// TwinCAT 3 PLC project Sample02
// ProgramVersion: 3.1.0.8
// libraries:
//   Tc2_Standard, * (Beckhoff Automation GmbH)
//   Tc2_System, * (Beckhoff Automation GmbH)
//   Tc2_Utilities, * (Beckhoff Automation GmbH)
//   Tc3_Interfaces, * (Beckhoff Automation GmbH)
//   Tc3_MemMan, * (Beckhoff Automation GmbH)
//   Tc3_Module, * (Beckhoff Automation GmbH)
// project tree:
//   / PlcTask.TcTTO (not stored)
//   POUs/ FB_AbstractLoggerFactory.TcPOU (not stored), FB_CsvLogger.TcPOU (not stored), FB_FileLoggerFactory.TcPOU, FB_Logger.TcPOU, FB_TxtLogger.TcPOU (not stored), FB_XmlLogger.TcPOU (not stored), ILogger.TcIO (not stored), MAIN.TcPOU
// real-time tasks:
//   TASK PlcTask: cycle T#10ms, priority 20, ADS port 350

// ---- POUs/FB_FileLoggerFactory.TcPOU
FUNCTION_BLOCK INTERNAL FB_FileLoggerFactory EXTENDS FB_AbstractLoggerFactory
VAR
	pTxtLogger  : POINTER TO FB_TxtLogger;
	pCsvLogger  : POINTER TO FB_CsvLogger;
	pXmlLogger  : POINTER TO FB_XmlLogger;
    ipLogger    : ILogger := 0;
END_VAR

METHOD FB_init : BOOL
VAR_INPUT
    bInitRetains  : BOOL; // if TRUE, the retain variables are initialized (warm start / cold start)
    bInCopyCode   : BOOL;  // if TRUE, the instance afterwards gets moved into the copy code (online change)
    sFilename     : STRING;
END_VAR
VAR
    sFilenameExtension : STRING;
END_VAR
sFilenameExtension := F_ToLCase(RIGHT(sFilename, 3));
IF (sFilenameExtension = 'txt') THEN
    pTxtLogger := __NEW(FB_TxtLogger);
    ipLogger := pTxtLogger^;
ELSIF (sFilenameExtension = 'csv') THEN
    pCsvLogger := __NEW(FB_CsvLogger);
    ipLogger := pCsvLogger^;
ELSIF (sFilenameExtension = 'xml') THEN
    pXmlLogger := __NEW(FB_XmlLogger);
    ipLogger := pXmlLogger^;
ELSE
    ipLogger := 0;
END_IF
END_METHOD

METHOD PUBLIC GetLogger : ILogger
VAR_INPUT
END_VAR
GetLogger := ipLogger;
END_METHOD

METHOD FB_exit : BOOL
VAR_INPUT
	bInCopyCode : BOOL; // if TRUE, the exit method is called for exiting an instance that is copied afterwards (online change).
END_VAR
IF (pTxtLogger <> 0) THEN
	__DELETE(pTxtLogger);
	pTxtLogger := 0;
END_IF

IF (pCsvLogger <> 0) THEN
	__DELETE(pCsvLogger);
	pCsvLogger := 0;
END_IF

IF (pXmlLogger <> 0) THEN
	__DELETE(pXmlLogger);
	pXmlLogger := 0;
END_IF
END_METHOD

END_FUNCTION_BLOCK

// ---- POUs/FB_Logger.TcPOU
FUNCTION_BLOCK PUBLIC FB_Logger
VAR
	ipLogger : ILogger;
END_VAR

METHOD PUBLIC Write : STRING
VAR_INPUT
	sMsg 		 : STRING;
END_VAR
Write := 'Error';
IF (ipLogger <> 0) THEN
	Write := ipLogger.Write(sMsg);
END_IF
END_METHOD

METHOD FB_init : BOOL
VAR_INPUT
	bInitRetains       : BOOL; // if TRUE, the retain variables are initialized (warm start / cold start)
	bInCopyCode        : BOOL;  // if TRUE, the instance afterwards gets moved into the copy code (online change)
	refLoggerFactory   : REFERENCE TO FB_AbstractLoggerFactory;
END_VAR
IF (__ISVALIDREF(refLoggerFactory)) THEN
	ipLogger := refLoggerFactory.GetLogger();
ELSE
	ipLogger := 0;
END_IF
END_METHOD

END_FUNCTION_BLOCK

// ---- POUs/MAIN.TcPOU
PROGRAM MAIN
VAR
	fbFileLoggerFactory	  : FB_FileLoggerFactory('File.csv');
	refFileLoggerFactory  : REFERENCE TO FB_FileLoggerFactory := fbFileLoggerFactory;
	fbLogger 			  : FB_Logger(refFileLoggerFactory);	
	sRetMsg				  : STRING;
END_VAR

sRetMsg := fbLogger.Write('Hello');

END_PROGRAM
